# EPICS substitutions: iocs/MC11/db/autohome.substitutions
file "db/autohome.db"
{
pattern
{SYS,           DEV,                 PLC,  PORT  }
{"XF:06BM-ES",  "{SixC-Ax:VTTH}",    8,    P0    }
{"XF:06BM-ES",  "{SixC-Ax:VTH}",     9,    P0    }
{"XF:06BM-ES",  "{SixC-Ax:CHI}",     10,   P0    }
{"XF:06BM-ES",  "{SixC-Ax:PHI}",     11,   P0    }
{"XF:06BM-ES",  "{SixC-Ax:HTH}",     12,   P0    }
{"XF:06BM-ES",  "{SixC-Ax:HTTH}",    13,   P0    }
{"XF:06BM-ES",  "{SixC-Ax:ANAL}",    14,   P0    }
{"XF:06BM-ES",  "{SixC-Ax:DET}",     15,   P0    }
}
